FUNCTION_BLOCK F_ADD (* Adds two number values *)
  (* Standard: 61131-3; Classification: standard arithmetic function; Description: Copyright (c) 2011 TU Wien ACIN This program and the accompanying materials are made available under the terms of the Eclipse Public License 2.0 which is available at https://www.eclipse.org/legal/epl-2.0/ SPDX-License-Identifier: EPL-2.0 *)
  (* Version 3.0, 2025-04-14, Patrick Aigner, changed package *)
  (* Version 1.0, 2011-09-22, Monika Wenger, TU Wien ACIN *)
  PACKAGE iec61131::arithmetic;
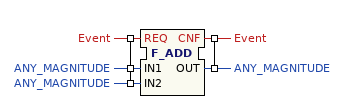
  EVENT_INPUT
    REQ WITH IN1, IN2; (* Normal Execution Request *)
  END_EVENT
  EVENT_OUTPUT
    CNF WITH OUT; (* Execution Confirmation *)
  END_EVENT
  VAR_INPUT
    IN1 : ANY_MAGNITUDE; (* First funtion input *)
    IN2 : ANY_MAGNITUDE; (* Second function input *)
  END_VAR
  VAR_OUTPUT
    OUT : ANY_MAGNITUDE; (* IN1 plus IN2 *)
  END_VAR
END_FUNCTION_BLOCK
